FUNCTION_BLOCK BACnetSubscribeUnconfirmedCOV (* Service Interface Function Block Type *)
  (* Standard: 61499-2 *)
  (* Version 1.0, 2020-01-18, root *)
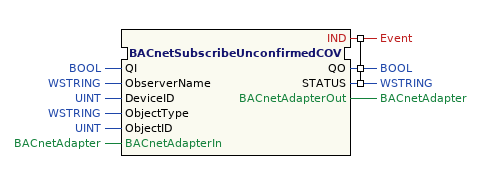
  EVENT_OUTPUT
    IND WITH QO, STATUS; (* Indication from Resource *)
  END_EVENT
  VAR_INPUT
    QI : BOOL; (* Event Input Qualifier *)
    ObserverName : WSTRING; (* Name of the Observer FB *)
    DeviceID : UINT; (* Identifier of the remote Device *)
    ObjectType : WSTRING; (* Object type of the target object *)
    ObjectID : UINT; (* Identifier of the target object *)
  END_VAR
  VAR_OUTPUT
    QO : BOOL; (* Event Output Qualifier *)
    STATUS : WSTRING; (* Service Status *)
  END_VAR
  SOCKETS
    BACnetAdapterIn : BACnetAdapter; (* BACnet adapter socket *)
  END_SOCKETS
  PLUGS
    BACnetAdapterOut : BACnetAdapter; (* BACnet adapter plug *)
  END_PLUGS
END_FUNCTION_BLOCK
